FUNCTION_BLOCK UR2 (* Tamplate for a simple Basic Function Block Type *)
  (* Standard: 61499-2 *)
  (* Version 0.0, 2018-01-29, 4DIAC-IDE, 4DIAC-Consortium *)
  (* Version 1.0, 2016-05-26, AZ, fortiss GmbH *)
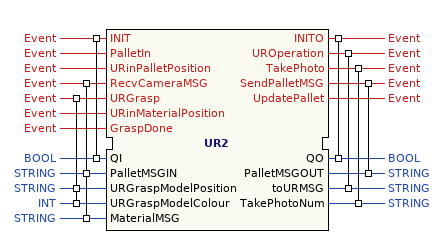
  EVENT_INPUT
    INIT WITH QI; (* Initialization Request *)
    PalletIn; (* Normal Execution Request *)
    URinPalletPosition;
    RecvCameraMSG WITH PalletMSGIN, MaterialMSG;
    URGrasp WITH URGraspModelPosition, URGraspModelColour;
    URinMaterialPosition;
    GraspDone;
  END_EVENT
  EVENT_OUTPUT
    INITO WITH QO; (* Initialization Confirm *)
    UROperation WITH toURMSG; (* Execution Confirmation *)
    TakePhoto WITH TakePhotoNum;
    SendPalletMSG WITH PalletMSGOUT;
    UpdatePallet;
  END_EVENT
  VAR_INPUT
    QI : BOOL; (* Input event qualifier *)
    PalletMSGIN : STRING;
    URGraspModelPosition : STRING;
    URGraspModelColour : INT;
    MaterialMSG : STRING;
  END_VAR
  VAR_OUTPUT
    QO : BOOL; (* Output event qualifier *)
    PalletMSGOUT : STRING;
    toURMSG : STRING;
    TakePhotoNum : STRING;
  END_VAR
  VAR
    color : INT; (* Internal Variable *)
    isMSGofPallet : BOOL; (* Internal Variable *)
    isExist : BOOL; (* Internal Variable *)
  END_VAR
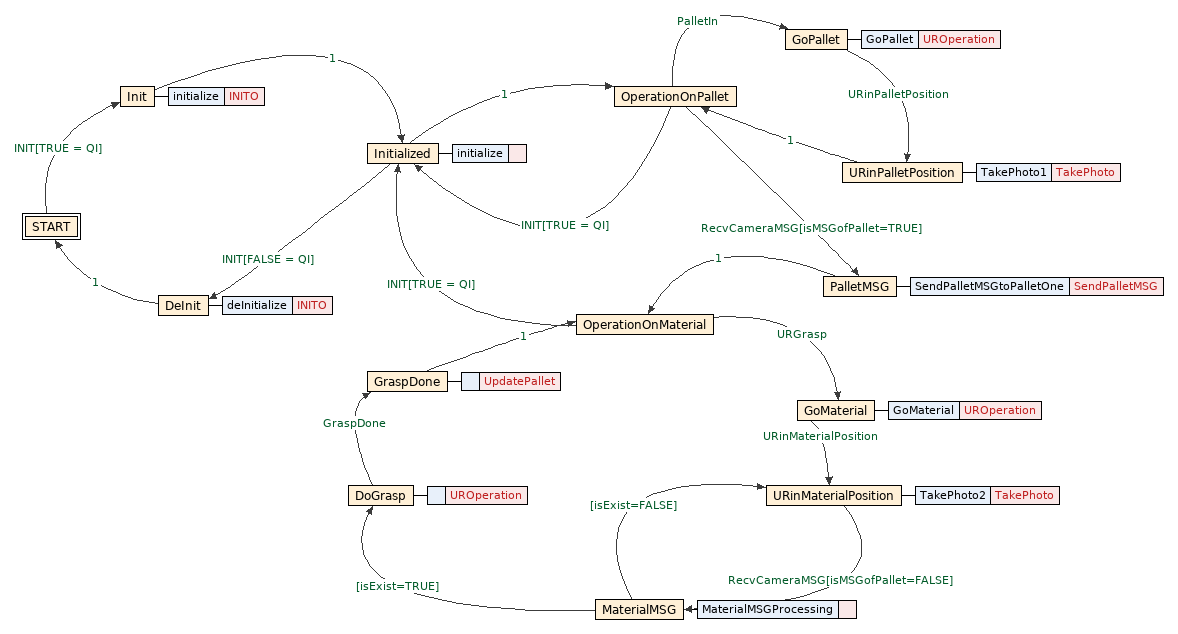
  EC_STATES
    START; (* Initial State *)
    Init : initialize -> INITO; (* Initialization *)
    Initialized : initialize;
    DeInit : deInitialize -> INITO;
    OperationOnPallet;
    GoPallet : GoPallet -> UROperation;
    URinPalletPosition : TakePhoto1 -> TakePhoto;
    PalletMSG : SendPalletMSGtoPalletOne -> SendPalletMSG; (* pallet MSG processing *)
    OperationOnMaterial;
    GoMaterial : GoMaterial -> UROperation;
    URinMaterialPosition : TakePhoto2 -> TakePhoto;
    MaterialMSG : MaterialMSGProcessing;
    DoGrasp : -> UROperation;
    GraspDone : -> UpdatePallet;
  END_STATES
  EC_TRANSITIONS
    START TO Init := INIT[TRUE = QI];
    Init TO Initialized := 1;
    DeInit TO START := 1;
    Initialized TO DeInit := INIT[FALSE = QI];
    Initialized TO OperationOnPallet := 1;
    OperationOnPallet TO GoPallet := PalletIn;
    GoPallet TO URinPalletPosition := URinPalletPosition;
    URinPalletPosition TO OperationOnPallet := 1;
    OperationOnPallet TO PalletMSG := RecvCameraMSG[isMSGofPallet=TRUE];
    PalletMSG TO OperationOnMaterial := 1;
    OperationOnMaterial TO GoMaterial := URGrasp;
    GoMaterial TO URinMaterialPosition := URinMaterialPosition;
    URinMaterialPosition TO MaterialMSG := RecvCameraMSG[isMSGofPallet=FALSE];
    MaterialMSG TO DoGrasp := [isExist=TRUE];
    MaterialMSG TO URinMaterialPosition := [isExist=FALSE];
    DoGrasp TO GraspDone := GraspDone;
    GraspDone TO OperationOnMaterial := 1;
    OperationOnMaterial TO Initialized := INIT[TRUE = QI];
    OperationOnPallet TO Initialized := INIT[TRUE = QI];
  END_TRANSITIONS
  ALGORITHM initialize IN ST: (* Initialization algorithm *)
QO := QI;
color:=0;
isMSGofPallet:=true;
isExist:=true;
  END_ALGORITHM
  ALGORITHM deInitialize IN ST: (* Normally executed algorithm *)
QO := FALSE;
  END_ALGORITHM
  ALGORITHM normalOperation IN ST: (* new algorithm *)
QO := QI;

IF TRUE  = QI THEN
  (*  only perform normal operation of QI is true*)

END_IF;
  END_ALGORITHM
  ALGORITHM GoPallet IN ST: (* new algorithm *)
toURMSG:='p';
  END_ALGORITHM
  ALGORITHM TakePhoto1 IN ST: (* new algorithm *)
TakePhotoNum:=1;
  END_ALGORITHM
  ALGORITHM SendPalletMSGtoPalletOne IN ST: (* new algorithm *)
PalletMSGOUT:=PalletMSGIN;
isMSGofPallet:=FALSE;
  END_ALGORITHM
  ALGORITHM GoMaterial IN ST: (* new algorithm *)
toURMSG:=URGraspModelPosition;
color:=URGraspModelColour;
  END_ALGORITHM
  ALGORITHM MaterialMSGProcessing IN ST: (* new algorithm *)

  END_ALGORITHM
  ALGORITHM StartGrasp IN ST: (* new algorithm *)

  END_ALGORITHM
  ALGORITHM TakePhoto2 IN ST: (* new algorithm *)
TakePhotoNum:=1;
  END_ALGORITHM
END_FUNCTION_BLOCK
